// TIA Portal V20 export
TYPE "UDT_FormatMsg"
   STRUCT
      Id : DInt;
      Severity : Byte;
      Active : Bool;
   END_STRUCT;
END_TYPE
